PROGRAM MAIN
VAR
END_VAR

P1();
P_Task2();

END_PROGRAM

(* stored: Version 1.1.0.1, ProductVersion 3.1.4024.12
   POU MAIN: Id {7a2fd32f-e666-4690-a0f1-b76dfc5f4749}, SpecialFunc None *)
